SUBAPPLICATION AX_E_PERMIT_INVERT_4 (* 4-Kanal Invertiertes Event-Freigabe-Gate mit Adapter (AX_NOT_INIT + AX_E_PERMIT_4) *)
  (* Standard: 61499-2; Description: Copyright (c) 2026 Meisterschulen am Ostbahnhof This program and the accompanying materials are made available under the terms of the Eclipse Public License 2.0 which is available at https://www.eclipse.org/legal/epl-2.0/ SPDX-License-Identifier: EPL-2.0 *)
  (* Version 1.0, 2026-09-10, Franz Höpfinger, Meisterschulen am Ostbahnhof, initial implementation *)
  PACKAGE MyLib::sys;
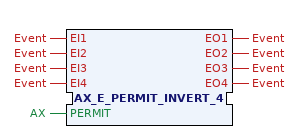
  EVENT_INPUT
    EI1; (* Event input channel 1 *)
    EI2; (* Event input channel 2 *)
    EI3; (* Event input channel 3 *)
    EI4; (* Event input channel 4 *)
  END_EVENT
  EVENT_OUTPUT
    EO1; (* Event output channel 1 *)
    EO2; (* Event output channel 2 *)
    EO3; (* Event output channel 3 *)
    EO4; (* Event output channel 4 *)
  END_EVENT
  SOCKETS
    PERMIT : adapter::types::unidirectional::AX; (* Invertiertes Freigabesignal *)
  END_SOCKETS
  FBS
    AX_NOT_INIT : adapter::booleanOperators::AX_NOT_INIT;
    AX_E_PERMIT_4 : adapter::events::unidirectional::AX_E_PERMIT_4;
  END_FBS
  EVENT_CONNECTIONS
    EI1 TO AX_E_PERMIT_4.EI1;
    AX_E_PERMIT_4.EO1 TO EO1;
    EI2 TO AX_E_PERMIT_4.EI2;
    AX_E_PERMIT_4.EO2 TO EO2;
    EI3 TO AX_E_PERMIT_4.EI3;
    AX_E_PERMIT_4.EO3 TO EO3;
    EI4 TO AX_E_PERMIT_4.EI4;
    AX_E_PERMIT_4.EO4 TO EO4;
  END_CONNECTIONS
  ADAPTER_CONNECTIONS
    PERMIT TO AX_NOT_INIT.IN;
    AX_NOT_INIT.OUT TO AX_E_PERMIT_4.PERMIT;
  END_CONNECTIONS
END_SUBAPPLICATION
